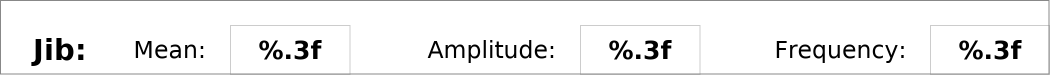
VISUALIZATION VISU_Sine_2  // 1050x75
    Textfield (230,25 120x50), "%.3f", text variable: G_Parameter.fJib_Mean
        OnMouseClick: write the text variable via InputWithLimits, min 0.1, max 0.7
    Textfield (110,25 120x50), "Mean:"
    Textfield (580,25 120x50), "%.3f", text variable: G_Parameter.fJib_Amplitude
        OnMouseClick: write the text variable via InputWithLimits, max 0.2
    Textfield (414,25 156x50), "Amplitude:"
    Textfield (930,25 120x50), "%.3f", text variable: G_Parameter.fJib_Frequency
        OnMouseClick: write the text variable via Edit
    Textfield (761,25 159x50), "Frequency:"
    Textfield (0,25 120x50), "Jib:"
END_VISUALIZATION

(* stored: Version 1.1.0.1
   Visu VISU_Sine_2: Id {985786b5-342b-4a99-a227-3867650ce40a} *)
